PROGRAM FB_Tank
VAR
END_VAR

END_PROGRAM

(* stored: Version 1.1.0.1, ProductVersion 3.1.4024.13
   POU FB_Tank: Id {7815b356-e436-492c-b1fa-45b05eddf80a}, SpecialFunc None *)
